# B&R Automation Studio project Servo
Automation Studio 4.12.2.93; technology packages: mapp 5.23.1, mappMotion 5.23.1, mappView 5.23.0

## Configuration Config1

CPU X20CP1586, AutomationRuntime B4.93, Build 4.1.2, Vc V4.72.6

### Hardware
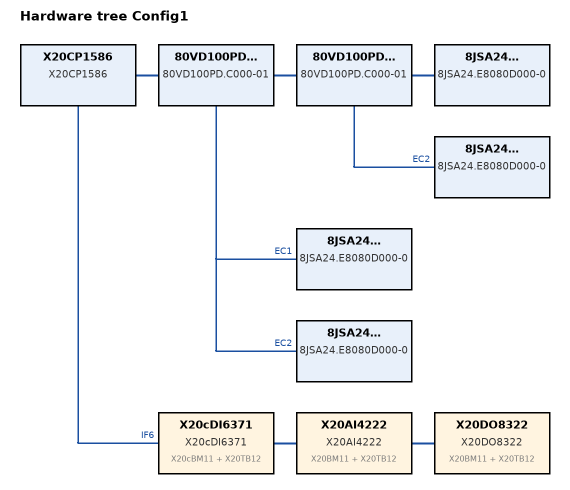
```
80VD100PD.C000-01 : 80VD100PD.C000-01 v2.5.0.0  [PLK1 -> 80VD100PD.C000-01a.PLK2 (NodeNumber=2) [Cable Type=PowerlinkCable, Length=10, Version=1.0.0.3]; EC1 -> 8JSA24.E8080D000-0.EC; EC2 -> 8JSA24.E8080D000-0a.EC; MT2 -> 8JSA24.E8080D000-0a.MT]
  DriveConfiguration/Module:
    McAcoposTypeID = AcoposMicroDConfig
    ActivateACOPOSSimulationOnPLC = 1
  DriveConfiguration/Channel[1]/RealAxis:
    AxisReference = gAxis_1
    MechanicalElementsIsInvisible = 0
  DriveConfiguration/Channel[1]/RealAxis/MechanicalElements/Gearbox:
    InputIsReadOnly = 0
    Input = 1
    OutputIsReadOnly = 0
    Output = 1
  DriveConfiguration/Channel[1]/RealAxis/MechanicalElements/RotaryToLinearTransformation:
    ReferenceDistanceIsReadOnly = 0
    ReferenceDistance = 1
  DriveConfiguration/Channel[1]/RealAxis/Controller:
    ModeIsReadOnly = 0
    Mode = PositionController
  DriveConfiguration/Channel[1]/RealAxis/Controller/Mode/Position:
    ProportionalGain = 50.0
    IntegrationTime = 0.0
    PredictionTime = 0.0004
    TotalDelayTime = 0.0004
  DriveConfiguration/Channel[1]/RealAxis/Controller/Mode/Speed:
    ProportionalGainIsReadOnly = 0
    ProportionalGain = 2.0
    IntegrationTimeIsReadOnly = 0
    IntegrationTime = 0.0
    FilterTimeIsReadOnly = 0
    FilterTime = 0.0
  DriveConfiguration/Channel[1]/RealAxis/Controller/Mode/LoopFilters:
    LoopFilterXIsReadOnly = 0
    LoopFilter1 = NotUsed
    LoopFilter2 = NotUsed
    LoopFilter3 = NotUsed
  DriveConfiguration/Channel[1]/RealAxis/Homing:
    ModeIsReadOnly = 0
    Mode = Direct
  DriveConfiguration/Channel[1]/RealAxis/Homing/Mode:
    Position = 0.0
    ReferencePulse = NotUsed
  DriveConfiguration/Channel[1]/RealAxis/Homing:
    RestorePositionVariable = 
  DriveConfiguration/Channel[1]/RealAxis/StopReaction:
    QuickstopIsReadOnly = 0
    Quickstop = DecelerationLimit
    DriveErrorIsReadOnly = 0
    DriveError = DecelerationLimit
  DriveConfiguration/Channel[1]/RealAxis/MovementErrorLimits:
    PositionError = 1.0
    VelocityErrorMonitoring = Automatic1
  DriveConfiguration/Channel[1]/RealAxis:
    JerkFilterIsReadOnly = 0
    JerkFilter = NotUsed
    ZeroVibrationFilter = NotUsed
  DriveConfiguration/Channel[1]/RealAxis/DigitalInputs/HomingSwitch:
    SourceIsReadOnly = 0
    Source = NotUsed
    Level = High
  DriveConfiguration/Channel[1]/RealAxis/DigitalInputs/PositiveLimitSwitch:
    SourceIsReadOnly = 0
    Source = NotUsed
    Level = High
  DriveConfiguration/Channel[1]/RealAxis/DigitalInputs/NegativeLimitSwitch:
    SourceIsReadOnly = 0
    Source = NotUsed
    Level = High
  DriveConfiguration/Channel[1]/RealAxis/DigitalInputs/Trigger1:
    Source = X2Trigger1
    Level = High
  DriveConfiguration/Channel[1]/RealAxis/DigitalInputs/Trigger2:
    Source = X2Trigger2
    Level = High
  DriveConfiguration/Channel[1]/RealAxis/DigitalInputs/Quickstop:
    Input = Trigger2
  DriveConfiguration/Channel[1]/RealAxis/Simulation:
    SimulationModeOnPLC = SetValueGeneration
    SimulationModeOnACOPOS = NotUsed
  DriveConfiguration/Channel[2]/RealAxis:
    AxisReference = gAxis_2
    MechanicalElementsIsInvisible = 0
  DriveConfiguration/Channel[2]/RealAxis/MechanicalElements/Gearbox:
    InputIsReadOnly = 0
    Input = 1
    OutputIsReadOnly = 0
    Output = 1
  DriveConfiguration/Channel[2]/RealAxis/MechanicalElements/RotaryToLinearTransformation:
    ReferenceDistanceIsReadOnly = 0
    ReferenceDistance = 1
  DriveConfiguration/Channel[2]/RealAxis/Controller:
    ModeIsReadOnly = 0
    Mode = PositionController
  DriveConfiguration/Channel[2]/RealAxis/Controller/Mode/Position:
    ProportionalGain = 50.0
    IntegrationTime = 0.0
    PredictionTime = 0.0004
    TotalDelayTime = 0.0004
  DriveConfiguration/Channel[2]/RealAxis/Controller/Mode/Speed:
    ProportionalGainIsReadOnly = 0
    ProportionalGain = 2.0
    IntegrationTimeIsReadOnly = 0
    IntegrationTime = 0.0
    FilterTimeIsReadOnly = 0
    FilterTime = 0.0
  DriveConfiguration/Channel[2]/RealAxis/Controller/Mode/LoopFilters:
    LoopFilterXIsReadOnly = 0
    LoopFilter1 = NotUsed
    LoopFilter2 = NotUsed
    LoopFilter3 = NotUsed
  DriveConfiguration/Channel[2]/RealAxis/Homing:
    ModeIsReadOnly = 0
    Mode = Direct
  DriveConfiguration/Channel[2]/RealAxis/Homing/Mode:
    Position = 0.0
    ReferencePulse = NotUsed
  DriveConfiguration/Channel[2]/RealAxis/Homing:
    RestorePositionVariable = 
  DriveConfiguration/Channel[2]/RealAxis/StopReaction:
    QuickstopIsReadOnly = 0
    Quickstop = DecelerationLimit
    DriveErrorIsReadOnly = 0
    DriveError = DecelerationLimit
  DriveConfiguration/Channel[2]/RealAxis/MovementErrorLimits:
    PositionError = 1.0
    VelocityErrorMonitoring = Automatic1
  DriveConfiguration/Channel[2]/RealAxis:
    JerkFilterIsReadOnly = 0
    JerkFilter = NotUsed
    ZeroVibrationFilter = NotUsed
  DriveConfiguration/Channel[2]/RealAxis/DigitalInputs/HomingSwitch:
    SourceIsReadOnly = 0
    Source = NotUsed
    Level = High
  DriveConfiguration/Channel[2]/RealAxis/DigitalInputs/PositiveLimitSwitch:
    SourceIsReadOnly = 0
    Source = NotUsed
    Level = High
  DriveConfiguration/Channel[2]/RealAxis/DigitalInputs/NegativeLimitSwitch:
    SourceIsReadOnly = 0
    Source = NotUsed
    Level = High
  DriveConfiguration/Channel[2]/RealAxis/DigitalInputs/Trigger1:
    Source = X2Trigger1
    Level = High
  DriveConfiguration/Channel[2]/RealAxis/DigitalInputs/Trigger2:
    Source = X2Trigger2
    Level = High
  DriveConfiguration/Channel[2]/RealAxis/DigitalInputs/Quickstop:
    Input = Trigger2
  DriveConfiguration/Channel[2]/RealAxis/Simulation:
    SimulationModeOnPLC = SetValueGeneration
    SimulationModeOnACOPOS = NotUsed
80VD100PD.C000-01a : 80VD100PD.C000-01 v2.5.0.0  [PLK1 -> X20CP1586.IF3 (NodeNumber=3) [Cable Type=PowerlinkCable, Length=10, Version=1.0.0.3]; PLK2 -> 80VD100PD.C000-01.PLK1 (NodeNumber=3) [Cable Type=PowerlinkCable, Length=10, Version=1.0.0.3]; EC1 -> 8JSA24.E8080D000-0b.EC; EC2 -> 8JSA24.E8080D000-0c.EC; MT2 -> 8JSA24.E8080D000-0c.MT]
  DriveConfiguration/Module:
    McAcoposTypeID = AcoposMicroDConfig
    ActivateACOPOSSimulationOnPLC = 1
  DriveConfiguration/Channel[1]/RealAxis:
    AxisReference = gAxis_3
    MechanicalElementsIsInvisible = 0
  DriveConfiguration/Channel[1]/RealAxis/MechanicalElements/Gearbox:
    InputIsReadOnly = 0
    Input = 1
    OutputIsReadOnly = 0
    Output = 1
  DriveConfiguration/Channel[1]/RealAxis/MechanicalElements/RotaryToLinearTransformation:
    ReferenceDistanceIsReadOnly = 0
    ReferenceDistance = 1
  DriveConfiguration/Channel[1]/RealAxis/Controller:
    ModeIsReadOnly = 0
    Mode = PositionController
  DriveConfiguration/Channel[1]/RealAxis/Controller/Mode/Position:
    ProportionalGain = 50.0
    IntegrationTime = 0.0
    PredictionTime = 0.0004
    TotalDelayTime = 0.0004
  DriveConfiguration/Channel[1]/RealAxis/Controller/Mode/Speed:
    ProportionalGainIsReadOnly = 0
    ProportionalGain = 2.0
    IntegrationTimeIsReadOnly = 0
    IntegrationTime = 0.0
    FilterTimeIsReadOnly = 0
    FilterTime = 0.0
  DriveConfiguration/Channel[1]/RealAxis/Controller/Mode/LoopFilters:
    LoopFilterXIsReadOnly = 0
    LoopFilter1 = NotUsed
    LoopFilter2 = NotUsed
    LoopFilter3 = NotUsed
  DriveConfiguration/Channel[1]/RealAxis/Homing:
    ModeIsReadOnly = 0
    Mode = Direct
  DriveConfiguration/Channel[1]/RealAxis/Homing/Mode:
    Position = 0.0
    ReferencePulse = Used
  DriveConfiguration/Channel[1]/RealAxis/Homing/Mode/ReferencePulse:
    HomingVelocity = 0.5
    Acceleration = 50.0
    HomingDirection = Positive
    KeepDirection = No
    ReferencePulseBlockingDistance = 0.0
  DriveConfiguration/Channel[1]/RealAxis/Homing:
    RestorePositionVariable = 
  DriveConfiguration/Channel[1]/RealAxis/StopReaction:
    QuickstopIsReadOnly = 0
    Quickstop = DecelerationLimit
    DriveErrorIsReadOnly = 0
    DriveError = DecelerationLimit
  DriveConfiguration/Channel[1]/RealAxis/MovementErrorLimits:
    PositionError = 1.0
    VelocityErrorMonitoring = Automatic1
  DriveConfiguration/Channel[1]/RealAxis:
    JerkFilterIsReadOnly = 0
    JerkFilter = NotUsed
    ZeroVibrationFilter = NotUsed
  DriveConfiguration/Channel[1]/RealAxis/DigitalInputs/HomingSwitch:
    SourceIsReadOnly = 0
    Source = NotUsed
    Level = High
  DriveConfiguration/Channel[1]/RealAxis/DigitalInputs/PositiveLimitSwitch:
    SourceIsReadOnly = 0
    Source = NotUsed
    Level = High
  DriveConfiguration/Channel[1]/RealAxis/DigitalInputs/NegativeLimitSwitch:
    SourceIsReadOnly = 0
    Source = NotUsed
    Level = High
  DriveConfiguration/Channel[1]/RealAxis/DigitalInputs/Trigger1:
    Source = X2Trigger1
    Level = High
  DriveConfiguration/Channel[1]/RealAxis/DigitalInputs/Trigger2:
    Source = X2Trigger2
    Level = High
  DriveConfiguration/Channel[1]/RealAxis/DigitalInputs/Quickstop:
    Input = Trigger2
  DriveConfiguration/Channel[1]/RealAxis/Simulation:
    SimulationModeOnPLC = SetValueGeneration
    SimulationModeOnACOPOS = NotUsed
  DriveConfiguration/Channel[2]/RealAxis:
    AxisReference = gAxis_4
    MechanicalElementsIsInvisible = 0
  DriveConfiguration/Channel[2]/RealAxis/MechanicalElements/Gearbox:
    InputIsReadOnly = 0
    Input = 1
    OutputIsReadOnly = 0
    Output = 1
  DriveConfiguration/Channel[2]/RealAxis/MechanicalElements/RotaryToLinearTransformation:
    ReferenceDistanceIsReadOnly = 0
    ReferenceDistance = 1
  DriveConfiguration/Channel[2]/RealAxis/Controller:
    ModeIsReadOnly = 0
    Mode = PositionController
  DriveConfiguration/Channel[2]/RealAxis/Controller/Mode/Position:
    ProportionalGain = 50.0
    IntegrationTime = 0.0
    PredictionTime = 0.0004
    TotalDelayTime = 0.0004
  DriveConfiguration/Channel[2]/RealAxis/Controller/Mode/Speed:
    ProportionalGainIsReadOnly = 0
    ProportionalGain = 2.0
    IntegrationTimeIsReadOnly = 0
    IntegrationTime = 0.0
    FilterTimeIsReadOnly = 0
    FilterTime = 0.0
  DriveConfiguration/Channel[2]/RealAxis/Controller/Mode/LoopFilters:
    LoopFilterXIsReadOnly = 0
    LoopFilter1 = NotUsed
    LoopFilter2 = NotUsed
    LoopFilter3 = NotUsed
  DriveConfiguration/Channel[2]/RealAxis/Homing:
    ModeIsReadOnly = 0
    Mode = Direct
  DriveConfiguration/Channel[2]/RealAxis/Homing/Mode:
    Position = 0.0
    ReferencePulse = NotUsed
  DriveConfiguration/Channel[2]/RealAxis/Homing:
    RestorePositionVariable = 
  DriveConfiguration/Channel[2]/RealAxis/StopReaction:
    QuickstopIsReadOnly = 0
    Quickstop = DecelerationLimit
    DriveErrorIsReadOnly = 0
    DriveError = DecelerationLimit
  DriveConfiguration/Channel[2]/RealAxis/MovementErrorLimits:
    PositionError = 1.0
    VelocityErrorMonitoring = Automatic1
  DriveConfiguration/Channel[2]/RealAxis:
    JerkFilterIsReadOnly = 0
    JerkFilter = NotUsed
    ZeroVibrationFilter = NotUsed
  DriveConfiguration/Channel[2]/RealAxis/DigitalInputs/HomingSwitch:
    SourceIsReadOnly = 0
    Source = NotUsed
    Level = High
  DriveConfiguration/Channel[2]/RealAxis/DigitalInputs/PositiveLimitSwitch:
    SourceIsReadOnly = 0
    Source = NotUsed
    Level = High
  DriveConfiguration/Channel[2]/RealAxis/DigitalInputs/NegativeLimitSwitch:
    SourceIsReadOnly = 0
    Source = NotUsed
    Level = High
  DriveConfiguration/Channel[2]/RealAxis/DigitalInputs/Trigger1:
    Source = X2Trigger1
    Level = High
  DriveConfiguration/Channel[2]/RealAxis/DigitalInputs/Trigger2:
    Source = X2Trigger2
    Level = High
  DriveConfiguration/Channel[2]/RealAxis/DigitalInputs/Quickstop:
    Input = Trigger2
  DriveConfiguration/Channel[2]/RealAxis/Simulation:
    SimulationModeOnPLC = SetValueGeneration
    SimulationModeOnACOPOS = NotUsed
8JSA24.E8080D000-0 : 8JSA24.E8080D000-0 v1.0.6.30  [EC -> 80VD100PD.C000-01.EC1; MT -> 80VD100PD.C000-01.MT1]
8JSA24.E8080D000-0a : 8JSA24.E8080D000-0 v1.0.6.30  [EC -> 80VD100PD.C000-01.EC2; MT -> 80VD100PD.C000-01.MT2]
8JSA24.E8080D000-0b : 8JSA24.E8080D000-0 v1.0.6.30  [EC -> 80VD100PD.C000-01a.EC1; MT -> 80VD100PD.C000-01a.MT1]
8JSA24.E8080D000-0c : 8JSA24.E8080D000-0 v1.0.6.30  [EC -> 80VD100PD.C000-01a.EC2; MT -> 80VD100PD.C000-01a.MT2]
X20AI4222 : X20AI4222 v1.2.0.0  [SS1 -> X20TB12b.SS; SL -> X20BM11a.SL1]
X20BM11 : X20BM11 v1.1.0.0  [X2X1 -> X20BM11a.X2X2]
X20BM11a : X20BM11 v1.1.0.0  [X2X1 -> X20cBM11.X2X2]
X20CP1586 : X20CP1586 v1.10.0.0
  Connector IF2:
    ActivateDevice = 1
  ConfigurationID = Servo_Config1
  Simulation = 1
  VolatileGlobalPvSize = 655350
  TimerDeviceType = EPLX2X
  TimerDevice = X20CP1586.IF3
  TaskClassIdleTime = 2000
  Cyclic1Duration = 8000
  Cyclic1Tolerance = 0
  Cyclic1Stack = 35563
  FileDevice1
  FileDeviceName1 = CF
  FileDevicePath1 = C:\history
  ActivateOpcUa = 1
  OpcUaInformationModels_PV_Version = 1
X20DO8322 : X20DO8322 v1.5.0.0  [SS1 -> X20TB12a.SS; SL -> X20BM11.SL1]
X20TB12 : X20TB12 v1.0.0.0
X20TB12a : X20TB12 v1.0.0.0
X20TB12b : X20TB12 v1.0.0.0
X20cBM11 : X20cBM11 v1.1.0.0  [X2X1 -> X20CP1586.IF6]
X20cDI6371 : X20cDI6371 v1.2.0.0  [SS1 -> X20TB12.SS; SL -> X20cBM11.SL1]
```

### Config_1.axis - X20CP1586/mappMotion/Config_1.axis
```
Element gAxis_1 (Type=axis)
  BaseTypeIsReadOnly = 0
  BaseType = LinearBounded
    MeasurementUnit = 5066068
    MeasurementResolutionIsReadOnly = 0
    MeasurementResolution = 0.01
    CountDirectionIsReadOnly = 0
    CountDirection = Standard
  MovementLimitsIsReadOnly = 0
  MovementLimits = Internal
    Position:
      LowerLimitMin = -1.79769313486231E308
      UpperLimitMax = 1.79769313486231E308
      LowerLimit = -100000
      UpperLimit = 100000
    VelocityIsReadOnly = 0
    Velocity:
      VelocityMax = 3.4E38
      Velocity = 10
    AccelerationIsReadOnly = 0
    Acceleration:
      AccelerationMax = 3.4E38
      Acceleration = 50
    DecelerationIsReadOnly = 0
    Deceleration:
      DecelerationMax = 3.4E38
      Deceleration = 50.0
  Alarms = None
```

### Config_2.axis - X20CP1586/mappMotion/Config_2.axis
```
Element gAxis_2 (Type=axis)
  BaseTypeIsReadOnly = 0
  BaseType = LinearBounded
    MeasurementUnit = 5066068
    MeasurementResolutionIsReadOnly = 0
    MeasurementResolution = 0.01
    CountDirectionIsReadOnly = 0
    CountDirection = Standard
  MovementLimitsIsReadOnly = 0
  MovementLimits = Internal
    Position:
      LowerLimitMin = -1.79769313486231E308
      UpperLimitMax = 1.79769313486231E308
      LowerLimit = -1000.0
      UpperLimit = 1000.0
    VelocityIsReadOnly = 0
    Velocity:
      VelocityMax = 3.4E38
      Velocity = 10.0
    AccelerationIsReadOnly = 0
    Acceleration:
      AccelerationMax = 3.4E38
      Acceleration = 50.0
    DecelerationIsReadOnly = 0
    Deceleration:
      DecelerationMax = 3.4E38
      Deceleration = 50.0
  Alarms = None
```

### Config_3.axis - X20CP1586/mappMotion/Config_3.axis
```
Element gAxis_3 (Type=axis)
  BaseTypeIsReadOnly = 0
  BaseType = LinearBounded
    MeasurementUnit = 5066068
    MeasurementResolutionIsReadOnly = 0
    MeasurementResolution = 0.01
    CountDirectionIsReadOnly = 0
    CountDirection = Standard
  MovementLimitsIsReadOnly = 0
  MovementLimits = Internal
    Position:
      LowerLimitMin = -1.79769313486231E308
      UpperLimitMax = 1.79769313486231E308
      LowerLimit = -1000.0
      UpperLimit = 1000.0
    VelocityIsReadOnly = 0
    Velocity:
      VelocityMax = 3.4E38
      Velocity = 10.0
    AccelerationIsReadOnly = 0
    Acceleration:
      AccelerationMax = 3.4E38
      Acceleration = 50.0
    DecelerationIsReadOnly = 0
    Deceleration:
      DecelerationMax = 3.4E38
      Deceleration = 50.0
  Alarms = None
```

### Config_4.axis - X20CP1586/mappMotion/Config_4.axis
```
Element gAxis_4 (Type=axis)
  BaseTypeIsReadOnly = 0
  BaseType = LinearBounded
    MeasurementUnit = 5066068
    MeasurementResolutionIsReadOnly = 0
    MeasurementResolution = 0.01
    CountDirectionIsReadOnly = 0
    CountDirection = Standard
  MovementLimitsIsReadOnly = 0
  MovementLimits = Internal
    Position:
      LowerLimitMin = -1.79769313486231E308
      UpperLimitMax = 1.79769313486231E308
      LowerLimit = -1000.0
      UpperLimit = 1000.0
    VelocityIsReadOnly = 0
    Velocity:
      VelocityMax = 3.4E38
      Velocity = 10.0
    AccelerationIsReadOnly = 0
    Acceleration:
      AccelerationMax = 3.4E38
      Acceleration = 50.0
    DecelerationIsReadOnly = 0
    Deceleration:
      DecelerationMax = 3.4E38
      Deceleration = 50.0
  Alarms = None
```

### Config.mpalarmxcore - X20CP1586/mappServices/Config.mpalarmxcore
```
Element gAlarmXCore (Type=mpalarmxcore)
  mapp.AlarmX.Core.Configuration:
    [0]:
      Name = Weedicide
      Message = {&LimitText}
      Code = 1000
      Severity = 10
      Behavior = LevelMonitoring
        Monitoring:
          MonitoredPV = ::Float
          LowLimitEnable = Static
            Limit = 50
            LimitText = weedicide remaining : below 50%
            LowLowLimitEnable = Static
              Limit = 16
              LimitText = weedicide remaining: critical below 15%
          HighLimitEnable = Static
            Limit = 50
            LimitText = weedicide remainig : above 50%
            HighHighLimitEnable = Static
              Limit = 99
              LimitText = Full capacity
    [1]:
      Name = Battery
      Message = {&LimitText}
      Code = 2000
      Severity = 20
      Behavior = LevelMonitoring
        Monitoring:
          MonitoredPV = ::Battery
          LowLimitEnable = Static
            Limit = 50
            LimitText = Battery status:below  50%
            LowLowLimitEnable = Static
              Limit = 16
              LimitText = Battery status: Critical below 15%
          HighLimitEnable = Static
            Limit = 50
            LimitText = Battery status: above 50%
            HighHighLimitEnable = Static
              Limit = 99
              LimitText = Battery status: fully charged 100%
```

## Logical view

Binary libraries used (declarations not repeated): operator, runtime, astime, AsIecCon, McBase, MpAxis, McAxis, MpBase, McAcpAx, standard, MpAlarmX, MpServer, MpRecipe 5.23.1, sys_lib

### Global.var - Global variables
```iecst
VAR
	RightAct : BOOL;
	Left_Proximity : BOOL;
	Right_Solenoid : BOOL;
	KEY : BOOL;
	Buzzer : BOOL;
	Right_Proximity : BOOL;
	Left_Solenoid : BOOL;
	LeftAct : BOOL;
	Proximity_1 : BOOL;
	Counter : INT := 0;
	Row : INT;
	LeftWheel_F : MpAxisBasic;
	LeftWheel_B : MpAxisBasic;
	RightWheel_F : MpAxisBasic;
	RightWheel_B : MpAxisBasic;
	AxisParameters : MpAxisBasicParType;
	State : BOOL := FALSE;
	MpAlarmXCore_0 : MpAlarmXCore;
	Pump : BOOL;
	MpAlarmXListUI_0 : MpAlarmXListUI;
	UIConnect : MpAlarmXListUIConnectType;
	MpAlarmXHistory_0 : MpAlarmXHistory;
	MpAlarmXHistoryUI_0 : MpAlarmXHistoryUI;
	UIConnectHistory : MpAlarmXHistoryUIConnectType;
	Battery : INT;
	Start : BOOL;
	Float : INT;
	totallane : INT;
	RowCheckL : BOOL;
	RowCheckR : BOOL;
	PumpPressure : INT := 0;
END_VAR
```


### Program Logical/servo (IEC)

#### Variables.var
```iecst
VAR
	TON_0 : TON;
	TOF_0 : TOF;
	TON_1 : TON;
END_VAR
```

#### Main.st
```iecst
PROGRAM _INIT
	LeftWheel_F.Enable := TRUE;
	LeftWheel_F.MpLink := ADR(gAxis_1);
	LeftWheel_F.Parameters := ADR(AxisParameters);

	LeftWheel_B.Enable := TRUE;
	LeftWheel_B.MpLink := ADR(gAxis_2);
	LeftWheel_B.Parameters := ADR(AxisParameters);

	RightWheel_F.Enable := TRUE;
	RightWheel_F.MpLink := ADR(gAxis_3);
	RightWheel_F.Parameters := ADR(AxisParameters);

	RightWheel_B.Enable := TRUE;
	RightWheel_B.MpLink := ADR(gAxis_4);
	RightWheel_B.Parameters := ADR(AxisParameters);
	MpAlarmXHistory_0.Export :=FALSE;
END_PROGRAM

PROGRAM _CYCLIC
	totallane;

	IF Start = TRUE AND Counter<>totallane THEN

		/////////////////////////////////////////////////////////////////////////////Robot Turning////////////////////////////////////////////////////////////////////////////////////////////////
		IF Proximity_1 = 1 AND NOT State THEN
			Counter := Counter+1;
			Pump := TRUE;
			Row := Counter MOD 2;
			IF Row=0 THEN
				RowCheckL:=TRUE;
				RowCheckR:=FALSE;
			ELSE
				RowCheckL:=FALSE;
				RowCheckR:=TRUE;
			END_IF
		ELSE
			TOF_0.IN := Proximity_1;
			Pump := FALSE;
			TOF_0.PT := T#5s;

		END_IF

		///////////////////////////////////////////////////////////////////Left Turning///////////////////////////////////////////////////////////////////////////////////////////////////////////
		IF Proximity_1 = 0 AND Row = 0 AND TOF_0.Q = TRUE THEN
			Pump := TRUE;
			IF LeftWheel_F.IsHomed = TRUE THEN
				LeftWheel_F.MoveVelocity := FALSE;
			END_IF
			IF LeftWheel_B.IsHomed = TRUE THEN
				LeftWheel_B.MoveVelocity := FALSE;
			END_IF
			IF RightWheel_F.IsHomed = TRUE THEN
				RightWheel_F.MoveVelocity := TRUE;
			END_IF
			IF RightWheel_B.IsHomed = TRUE THEN
				RightWheel_B.MoveVelocity := TRUE;
			END_IF

			////////////////////////////////////////////////////////////////////Right Turning////////////////////////////////////////////////////////////////////////////////////////////////
		ELSIF Proximity_1 = 0 AND Row = 1 AND TOF_0.Q = TRUE THEN
			Pump := TRUE;
			IF RightWheel_F.IsHomed = TRUE THEN
				RightWheel_F.MoveVelocity := FALSE;
			END_IF
			IF RightWheel_B.IsHomed = TRUE THEN
				RightWheel_B.MoveVelocity := FALSE;
			END_IF
			IF LeftWheel_F.IsHomed = TRUE THEN
				LeftWheel_F.MoveVelocity := TRUE;
			END_IF
			IF LeftWheel_B.IsHomed = TRUE THEN
				LeftWheel_B.MoveVelocity := TRUE;
			END_IF
	ELSIF Proximity_1 = 0 AND Row = 0 THEN
		IF LeftWheel_F.Info.ReadyToPowerOn = TRUE THEN
			LeftWheel_F.Power := TRUE;
			IF LeftWheel_F.PowerOn = TRUE THEN
				LeftWheel_F.Home := TRUE;
				IF LeftWheel_F.IsHomed = TRUE THEN
					LeftWheel_F.MoveVelocity := TRUE;
				END_IF
			END_IF
		END_IF
		IF LeftWheel_B.Info.ReadyToPowerOn = TRUE THEN
			LeftWheel_B.Power := TRUE;
			IF LeftWheel_B.PowerOn = TRUE THEN
				LeftWheel_B.Home := TRUE;
				IF LeftWheel_B.IsHomed = TRUE THEN
					LeftWheel_B.MoveVelocity := TRUE;
				END_IF
			END_IF
		END_IF

		IF RightWheel_F.Info.ReadyToPowerOn = TRUE THEN
			RightWheel_F.Power := TRUE;
			IF RightWheel_F.PowerOn = TRUE THEN
				RightWheel_F.Home := TRUE;
				IF RightWheel_F.IsHomed = TRUE THEN
					RightWheel_F.MoveVelocity := TRUE;
				END_IF
			END_IF
		END_IF
		IF RightWheel_B.Info.ReadyToPowerOn = TRUE THEN
			RightWheel_B.Power := TRUE;
			IF RightWheel_B.PowerOn = TRUE THEN
				RightWheel_B.Home := TRUE;
				IF RightWheel_B.IsHomed = TRUE THEN
					RightWheel_B.MoveVelocity := TRUE;
				END_IF
			END_IF
		END_IF

	ELSIF Proximity_1 = 0 AND Row = 1 THEN
		IF LeftWheel_F.Info.ReadyToPowerOn = TRUE THEN
			LeftWheel_F.Power := TRUE;
			IF LeftWheel_F.PowerOn = TRUE THEN
				LeftWheel_F.Home := TRUE;
				IF LeftWheel_F.IsHomed = TRUE THEN
					LeftWheel_F.MoveVelocity := TRUE;
				END_IF
			END_IF
			END_IF
		IF LeftWheel_B.Info.ReadyToPowerOn = TRUE THEN
			LeftWheel_B.Power := TRUE;
			IF LeftWheel_B.PowerOn = TRUE THEN
				LeftWheel_B.Home := TRUE;
				IF LeftWheel_B.IsHomed = TRUE THEN
					LeftWheel_B.MoveVelocity := TRUE;
				END_IF
			END_IF
		END_IF

		IF RightWheel_F.Info.ReadyToPowerOn = TRUE THEN
			RightWheel_F.Power := TRUE;
			IF RightWheel_F.PowerOn = TRUE THEN
				RightWheel_F.Home := TRUE;
				IF RightWheel_F.IsHomed = TRUE THEN
					RightWheel_F.MoveVelocity := TRUE;
				END_IF
			END_IF
		END_IF
		IF RightWheel_B.Info.ReadyToPowerOn = TRUE THEN
			RightWheel_B.Power := TRUE;
			IF RightWheel_B.PowerOn = TRUE THEN
				RightWheel_B.Home := TRUE;
				IF RightWheel_B.IsHomed = TRUE THEN
					RightWheel_B.MoveVelocity := TRUE;
				END_IF
			END_IF
		END_IF

	END_IF
	State := Proximity_1;
	ELSIF Start = FALSE OR Counter=totallane THEN
		Start:=FALSE;
		Counter:=0;
	IF LeftWheel_F.Info.ReadyToPowerOn = TRUE THEN
		LeftWheel_F.Power := FALSE;
		IF LeftWheel_F.PowerOn = TRUE THEN
			LeftWheel_F.Home := FALSE;
			IF LeftWheel_F.IsHomed = TRUE THEN
				LeftWheel_F.MoveVelocity := FALSE;
			END_IF
		END_IF
	END_IF
	IF LeftWheel_B.Info.ReadyToPowerOn = TRUE THEN
		LeftWheel_B.Power := FALSE;
		IF LeftWheel_B.PowerOn = TRUE THEN
			LeftWheel_B.Home := FALSE;
			IF LeftWheel_B.IsHomed = TRUE THEN
				LeftWheel_B.MoveVelocity := FALSE;
			END_IF
		END_IF
	END_IF
	IF RightWheel_F.Info.ReadyToPowerOn = TRUE THEN
		RightWheel_F.Power := FALSE;
		IF RightWheel_F.PowerOn = TRUE THEN
			RightWheel_F.Home := FALSE;
			IF RightWheel_F.IsHomed = TRUE THEN
				RightWheel_F.MoveVelocity := FALSE;
			END_IF
		END_IF
	END_IF
	IF RightWheel_B.Info.ReadyToPowerOn = TRUE THEN
		RightWheel_B.Power := FALSE;
		IF RightWheel_B.PowerOn = TRUE THEN
			RightWheel_B.Home := FALSE;
			IF RightWheel_B.IsHomed = TRUE THEN
				RightWheel_B.MoveVelocity := FALSE;
			END_IF
		END_IF
	END_IF
	END_IF
	////////////////////////////////////////////////////////////////////////////Left Sensor////////////////////////////////////////////////////////////////////////////////////////////////////
	IF Right_Proximity = 1 THEN
		Right_Solenoid := FALSE;
		RightAct := TRUE;
	ELSE
		//Rotate inside
		Right_Solenoid := TRUE;
		RightAct := FALSE;
	END_IF

	////////////////////////////////////////////////////////////////////////////Right Sensor////////////////////////////////////////////////////////////////////////////////////////////////////
	IF Left_Proximity = 1 THEN
		Left_Solenoid := FALSE;
		LeftAct := TRUE;
	ELSE
		//Rotate inside
		Left_Solenoid := TRUE;
		LeftAct := FALSE;
	END_IF

	/////////////////////////////////////////////////////////////////////////////Floatsensor value Float1 Float2//////////////////////////////////////////////////////////////////////////////////////////
	MpAlarmXCore_0.Enable := TRUE;
	MpAlarmXCore_0.MpLink := ADR(gAlarmXCore);
	MpAlarmXCore_0();

	MpAlarmXListUI_0.Enable:=TRUE;
	MpAlarmXListUI_0.MpLink:=ADR(gAlarmXCore);
	MpAlarmXListUI_0.UIConnect:=ADR(UIConnect);
	MpAlarmXListUI_0();
	////////////////////////////////////////////////////////////////////////////AlarmHistory/////////////////////////////////////////////////////////////////////////////////////////////////////
	MpAlarmXHistory_0.Enable := TRUE;
	MpAlarmXHistory_0.DeviceName := ADR('CF');
	MpAlarmXHistory_0.MpLink := ADR(gAlarmXHistory);
	MpAlarmXHistory_0();

	MpAlarmXHistoryUI_0.Enable :=TRUE;
	MpAlarmXHistoryUI_0.MpLink := ADR(gAlarmXHistory);
	MpAlarmXHistoryUI_0.UIConnect := ADR(UIConnectHistory);
	MpAlarmXHistoryUI_0();

	//MpAlarmXHistoryUI_0(MpLink :=ADR(gAlarmXHistory) , Enable := TRUE, ErrorReset := TRUE,UIConnect :=ADR(AlarmXHistoryUIConnect) );
	////////////////////////////////////////////////////////////////////////////Robot Identification/////////////////////////////////////////////////////////////////////////////////////////////
	IF KEY = TRUE THEN
		Buzzer := TRUE;
	ELSE
		Buzzer := FALSE;
	END_IF
	Battery;
	Float;

	/////////////////////////////////////////////////////////////////////////////Function call////////////////////////////////////////////////////////////////////////////////////////////////
	LeftWheel_F();
	LeftWheel_B();
	RightWheel_F();
	RightWheel_B();
	TOF_0();
	MpAlarmXCore_0();
END_PROGRAM

PROGRAM _EXIT

END_PROGRAM
```

- Visualisation Logical/mappView (not shown)

Listed in the project but not available here: Logical/Global.typ
